PROGRAM p04_latch
VAR
	M0: BOOL;
	M1: BOOL;
END_VAR

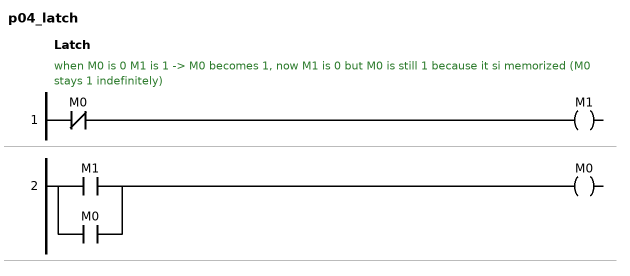
// NETWORK 1: Latch
// when M0 is 0 M1 is 1 -> M0 becomes 1, now M1 is 0 but M0 is still 1 because it si memorized (M0 stays 1 indefinitely)
M1 := NOT M0;

// NETWORK 2
M0 := M1 OR M0;

END_PROGRAM

(* stored: Version 1.1.0.1, ProductVersion 3.1.4024.13
   POU p04_latch: Id {258bf061-4f56-4924-b374-56259739d855}, SpecialFunc None *)
